// TIA Portal V19 export
DATA_BLOCK "DB_Arduino_Data"   // DB3
{ S7_Optimized_Access := 'FALSE' }
   VAR
      Read_Data : Array[1..120] of Word;
      Write_Data : Array[1..120] of Word;
   END_VAR
BEGIN
   Write_Data[1] := 16#B;
   Write_Data[2] := 16#E;
   Write_Data[3] := 16#0;
END_DATA_BLOCK
